# EPICS autosave request: support/delaygen-1-0-5/delaygenApp/Db/drvAsynCoherentSDG.req
$(P)$(R)Ch1outDelayStepAO
$(P)$(R)Ch2outDelayStepAO
$(P)$(R)Ch3outDelayStepAO
